// Mitsubishi GX Works2 project: BMA-PGM(V0.24)-20230412   PLC: Q06UDV

PROGRAM 02  // MANUAL
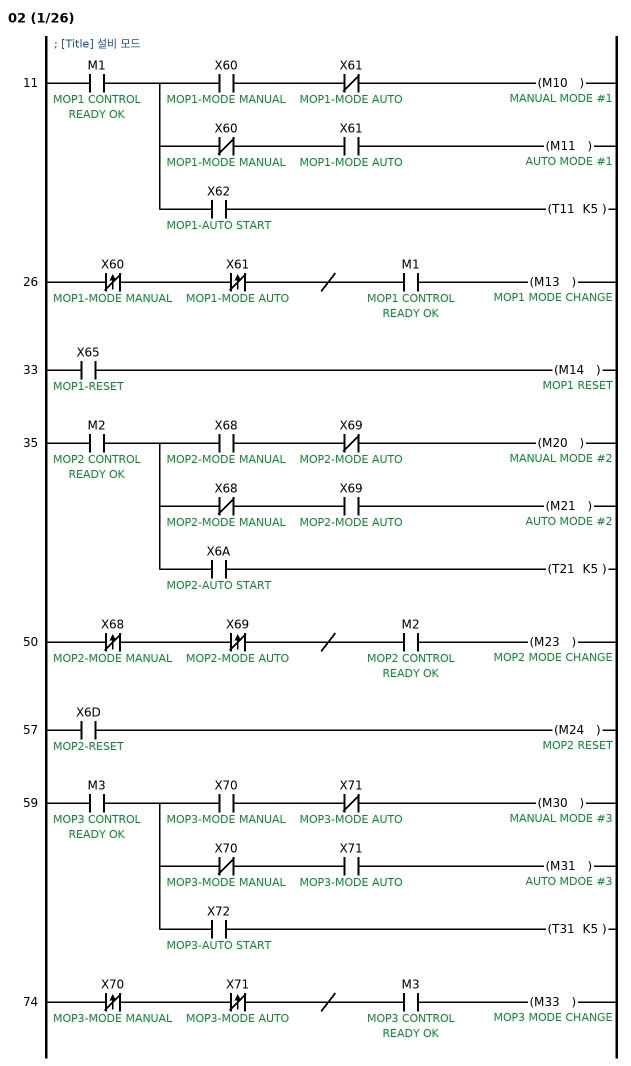
; [Title] 설비 모드
11    LD      M1  ; MOP1 CONTROL READY OK
      MPS
      AND     X60  ; MOP1-MODE MANUAL
      ANI     X61  ; MOP1-MODE AUTO
      OUT     M10  ; MANUAL MODE #1
      MRD
      ANI     X60  ; MOP1-MODE MANUAL
      AND     X61  ; MOP1-MODE AUTO
      OUT     M11  ; AUTO MODE #1
      MPP
      AND     X62  ; MOP1-AUTO START
      OUT     T11 K5
26    LDPI    X60  ; MOP1-MODE MANUAL
      ANDPI   X61  ; MOP1-MODE AUTO
      INV
      AND     M1  ; MOP1 CONTROL READY OK
      OUT     M13  ; MOP1 MODE CHANGE
33    LD      X65  ; MOP1-RESET
      OUT     M14  ; MOP1 RESET
35    LD      M2  ; MOP2 CONTROL READY OK
      MPS
      AND     X68  ; MOP2-MODE MANUAL
      ANI     X69  ; MOP2-MODE AUTO
      OUT     M20  ; MANUAL MODE #2
      MRD
      ANI     X68  ; MOP2-MODE MANUAL
      AND     X69  ; MOP2-MODE AUTO
      OUT     M21  ; AUTO MODE #2
      MPP
      AND     X6A  ; MOP2-AUTO START
      OUT     T21 K5
50    LDPI    X68  ; MOP2-MODE MANUAL
      ANDPI   X69  ; MOP2-MODE AUTO
      INV
      AND     M2  ; MOP2 CONTROL READY OK
      OUT     M23  ; MOP2 MODE CHANGE
57    LD      X6D  ; MOP2-RESET
      OUT     M24  ; MOP2 RESET
59    LD      M3  ; MOP3 CONTROL READY OK
      MPS
      AND     X70  ; MOP3-MODE MANUAL
      ANI     X71  ; MOP3-MODE AUTO
      OUT     M30  ; MANUAL MODE #3
      MRD
      ANI     X70  ; MOP3-MODE MANUAL
      AND     X71  ; MOP3-MODE AUTO
      OUT     M31  ; AUTO MDOE #3
      MPP
      AND     X72  ; MOP3-AUTO START
      OUT     T31 K5
74    LDPI    X70  ; MOP3-MODE MANUAL
      ANDPI   X71  ; MOP3-MODE AUTO
      INV
      AND     M3  ; MOP3 CONTROL READY OK
      OUT     M33  ; MOP3 MODE CHANGE
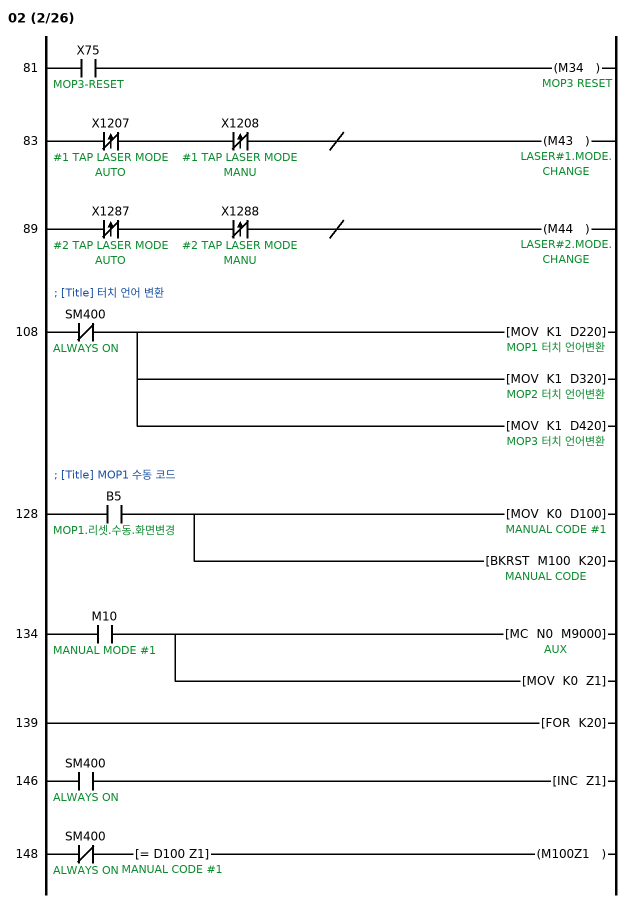
81    LD      X75  ; MOP3-RESET
      OUT     M34  ; MOP3 RESET
83    LDPI    X1207  ; #1 TAP LASER MODE AUTO
      ANDPI   X1208  ; #1 TAP LASER MODE MANU
      INV
      OUT     M43  ; LASER#1.MODE.CHANGE
89    LDPI    X1287  ; #2 TAP LASER MODE AUTO
      ANDPI   X1288  ; #2 TAP LASER MODE MANU
      INV
      OUT     M44  ; LASER#2.MODE.CHANGE
; [Title] 터치 언어 변환
108   LDI     SM400  ; ALWAYS ON
      MOV     K1 D220  ; MOP1 터치 언어변환
      MOV     K1 D320  ; MOP2 터치 언어변환
      MOV     K1 D420  ; MOP3 터치 언어변환
; [Title] MOP1 수동 코드
128   LD      B5  ; MOP1.리셋.수동.화면변경
      MOV     K0 D100  ; MANUAL CODE #1
      BKRST   M100 K20  ; MANUAL CODE
134   LD      M10  ; MANUAL MODE #1
      MC      N0 M9000  ; AUX
      MOV     K0 Z1
139   FOR     K20
        [note] 1~20
146   LD      SM400  ; ALWAYS ON
      INC     Z1
148   LDI     SM400  ; ALWAYS ON
      AND=    D100 Z1  ; MANUAL CODE #1
      OUT     M100Z1
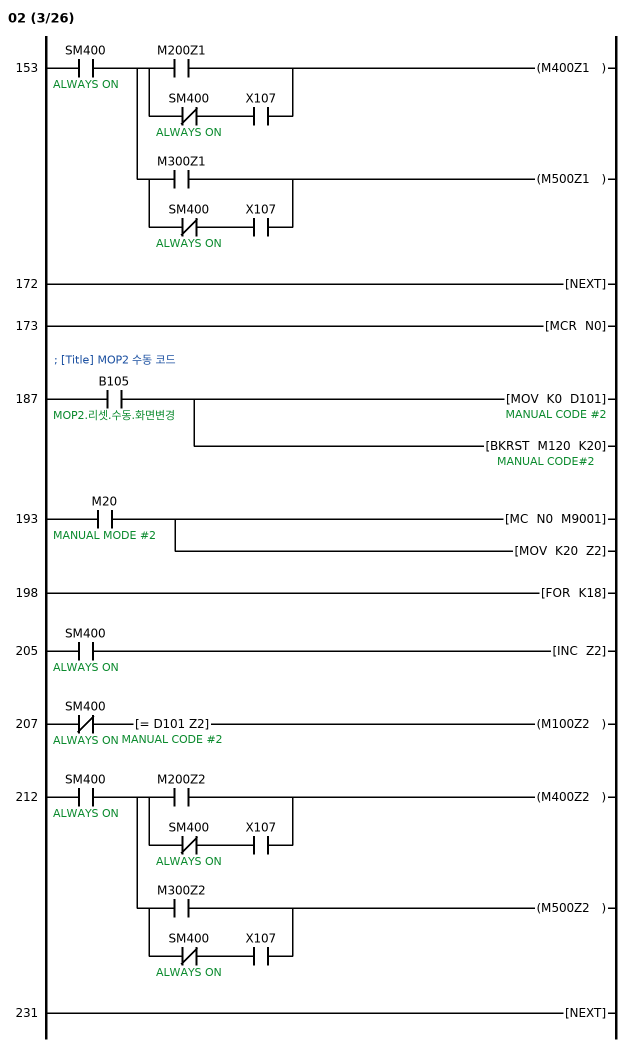
153   LD      SM400  ; ALWAYS ON
      MPS
      LD      M200Z1
      LDI     SM400  ; ALWAYS ON
      AND     X107
      ORB
      ANB
      OUT     M400Z1
      MPP
      LD      M300Z1
      LDI     SM400  ; ALWAYS ON
      AND     X107
      ORB
      ANB
      OUT     M500Z1
172   NEXT
173   MCR     N0
; [Title] MOP2 수동 코드
187   LD      B105  ; MOP2.리셋.수동.화면변경
      MOV     K0 D101  ; MANUAL CODE #2
      BKRST   M120 K20  ; MANUAL CODE#2
193   LD      M20  ; MANUAL MODE #2
      MC      N0 M9001
      MOV     K20 Z2
198   FOR     K18
        [note] 21~38
205   LD      SM400  ; ALWAYS ON
      INC     Z2
207   LDI     SM400  ; ALWAYS ON
      AND=    D101 Z2  ; MANUAL CODE #2
      OUT     M100Z2
212   LD      SM400  ; ALWAYS ON
      MPS
      LD      M200Z2
      LDI     SM400  ; ALWAYS ON
      AND     X107
      ORB
      ANB
      OUT     M400Z2
      MPP
      LD      M300Z2
      LDI     SM400  ; ALWAYS ON
      AND     X107
      ORB
      ANB
      OUT     M500Z2
231   NEXT
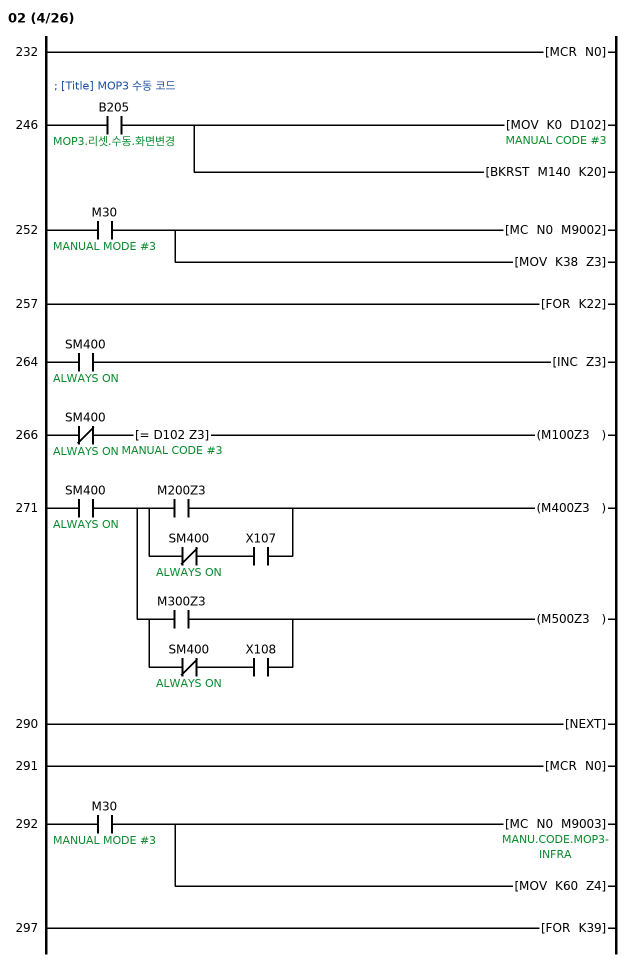
232   MCR     N0
; [Title] MOP3 수동 코드
246   LD      B205  ; MOP3.리셋.수동.화면변경
      MOV     K0 D102  ; MANUAL CODE #3
      BKRST   M140 K20
252   LD      M30  ; MANUAL MODE #3
      MC      N0 M9002
      MOV     K38 Z3
257   FOR     K22
        [note] 39~60
264   LD      SM400  ; ALWAYS ON
      INC     Z3
266   LDI     SM400  ; ALWAYS ON
      AND=    D102 Z3  ; MANUAL CODE #3
      OUT     M100Z3
271   LD      SM400  ; ALWAYS ON
      MPS
      LD      M200Z3
      LDI     SM400  ; ALWAYS ON
      AND     X107
      ORB
      ANB
      OUT     M400Z3
      MPP
      LD      M300Z3
      LDI     SM400  ; ALWAYS ON
      AND     X108
      ORB
      ANB
      OUT     M500Z3
290   NEXT
291   MCR     N0
292   LD      M30  ; MANUAL MODE #3
      MC      N0 M9003  ; MANU.CODE.MOP3-INFRA
      MOV     K60 Z4
297   FOR     K39
        [note] 61~99
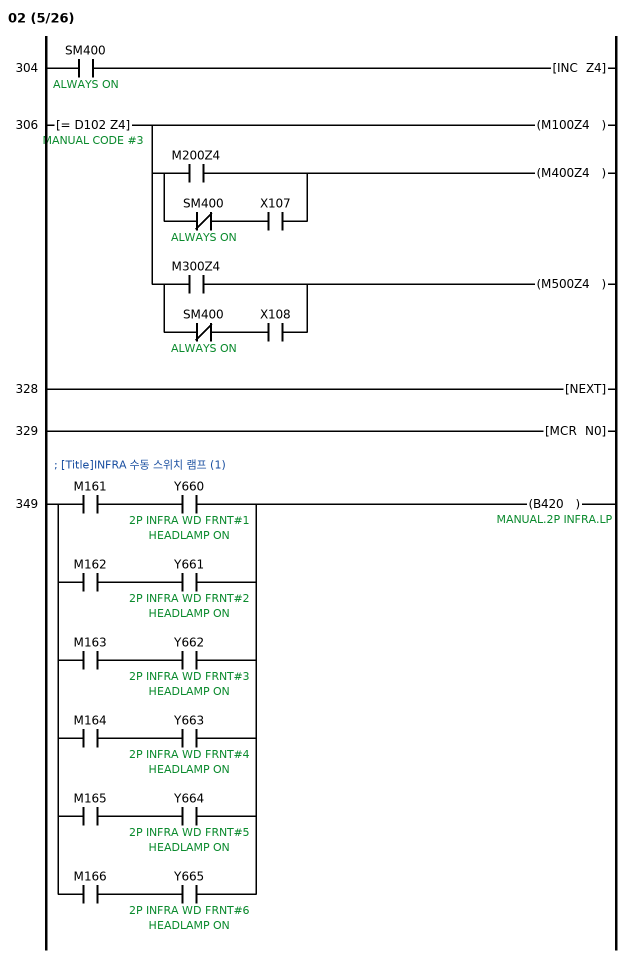
304   LD      SM400  ; ALWAYS ON
      INC     Z4
306   LD=     D102 Z4  ; MANUAL CODE #3
      OUT     M100Z4
      MPS
      LD      M200Z4
      LDI     SM400  ; ALWAYS ON
      AND     X107
      ORB
      ANB
      OUT     M400Z4
      MPP
      LD      M300Z4
      LDI     SM400  ; ALWAYS ON
      AND     X108
      ORB
      ANB
      OUT     M500Z4
328   NEXT
329   MCR     N0
; [Title]INFRA 수동 스위치 램프 (1)
349   LD      M161
      AND     Y660  ; 2P INFRA WD FRNT#1 HEADLAMP ON
      LD      M162
      AND     Y661  ; 2P INFRA WD FRNT#2 HEADLAMP ON
      ORB
      LD      M163
      AND     Y662  ; 2P INFRA WD FRNT#3 HEADLAMP ON
      ORB
      LD      M164
      AND     Y663  ; 2P INFRA WD FRNT#4 HEADLAMP ON
      ORB
      LD      M165
      AND     Y664  ; 2P INFRA WD FRNT#5 HEADLAMP ON
      ORB
      LD      M166
      AND     Y665  ; 2P INFRA WD FRNT#6 HEADLAMP ON
      ORB
      OUT     B420  ; MANUAL.2P INFRA.LP
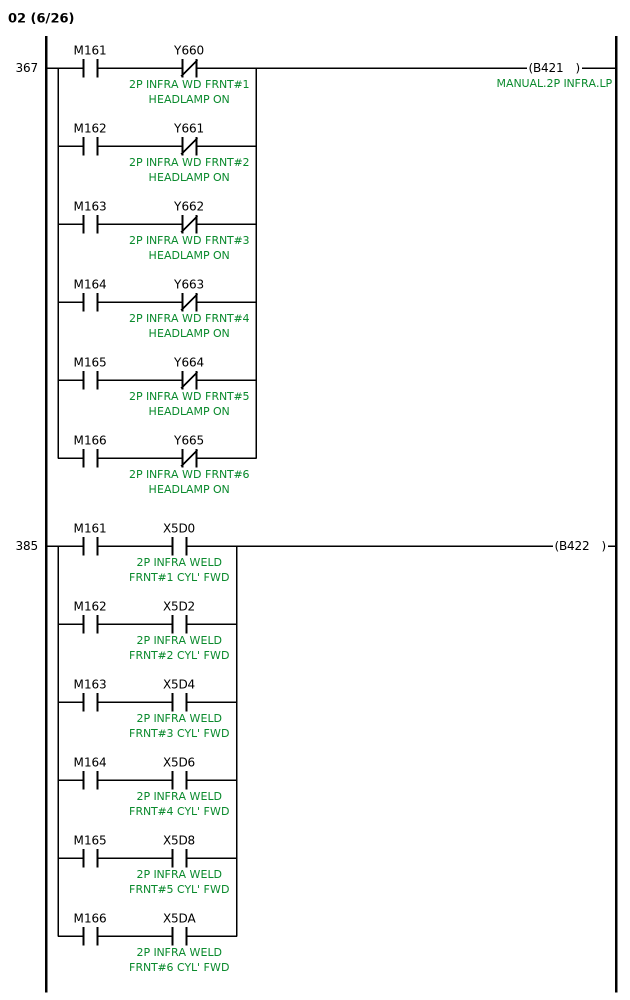
367   LD      M161
      ANI     Y660  ; 2P INFRA WD FRNT#1 HEADLAMP ON
      LD      M162
      ANI     Y661  ; 2P INFRA WD FRNT#2 HEADLAMP ON
      ORB
      LD      M163
      ANI     Y662  ; 2P INFRA WD FRNT#3 HEADLAMP ON
      ORB
      LD      M164
      ANI     Y663  ; 2P INFRA WD FRNT#4 HEADLAMP ON
      ORB
      LD      M165
      ANI     Y664  ; 2P INFRA WD FRNT#5 HEADLAMP ON
      ORB
      LD      M166
      ANI     Y665  ; 2P INFRA WD FRNT#6 HEADLAMP ON
      ORB
      OUT     B421  ; MANUAL.2P INFRA.LP
385   LD      M161
      AND     X5D0  ; 2P INFRA WELD FRNT#1 CYL' FWD
      LD      M162
      AND     X5D2  ; 2P INFRA WELD FRNT#2 CYL' FWD
      ORB
      LD      M163
      AND     X5D4  ; 2P INFRA WELD FRNT#3 CYL' FWD
      ORB
      LD      M164
      AND     X5D6  ; 2P INFRA WELD FRNT#4 CYL' FWD
      ORB
      LD      M165
      AND     X5D8  ; 2P INFRA WELD FRNT#5 CYL' FWD
      ORB
      LD      M166
      AND     X5DA  ; 2P INFRA WELD FRNT#6 CYL' FWD
      ORB
      OUT     B422
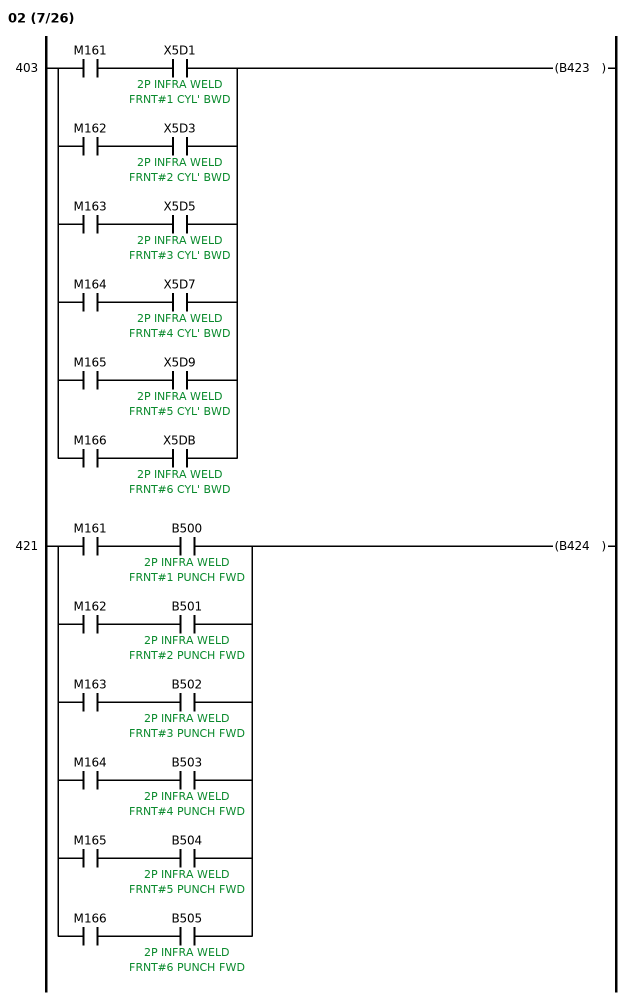
403   LD      M161
      AND     X5D1  ; 2P INFRA WELD FRNT#1 CYL' BWD
      LD      M162
      AND     X5D3  ; 2P INFRA WELD FRNT#2 CYL' BWD
      ORB
      LD      M163
      AND     X5D5  ; 2P INFRA WELD FRNT#3 CYL' BWD
      ORB
      LD      M164
      AND     X5D7  ; 2P INFRA WELD FRNT#4 CYL' BWD
      ORB
      LD      M165
      AND     X5D9  ; 2P INFRA WELD FRNT#5 CYL' BWD
      ORB
      LD      M166
      AND     X5DB  ; 2P INFRA WELD FRNT#6 CYL' BWD
      ORB
      OUT     B423
421   LD      M161
      AND     B500  ; 2P INFRA WELD FRNT#1 PUNCH FWD
      LD      M162
      AND     B501  ; 2P INFRA WELD FRNT#2 PUNCH FWD
      ORB
      LD      M163
      AND     B502  ; 2P INFRA WELD FRNT#3 PUNCH FWD
      ORB
      LD      M164
      AND     B503  ; 2P INFRA WELD FRNT#4 PUNCH FWD
      ORB
      LD      M165
      AND     B504  ; 2P INFRA WELD FRNT#5 PUNCH FWD
      ORB
      LD      M166
      AND     B505  ; 2P INFRA WELD FRNT#6 PUNCH FWD
      ORB
      OUT     B424
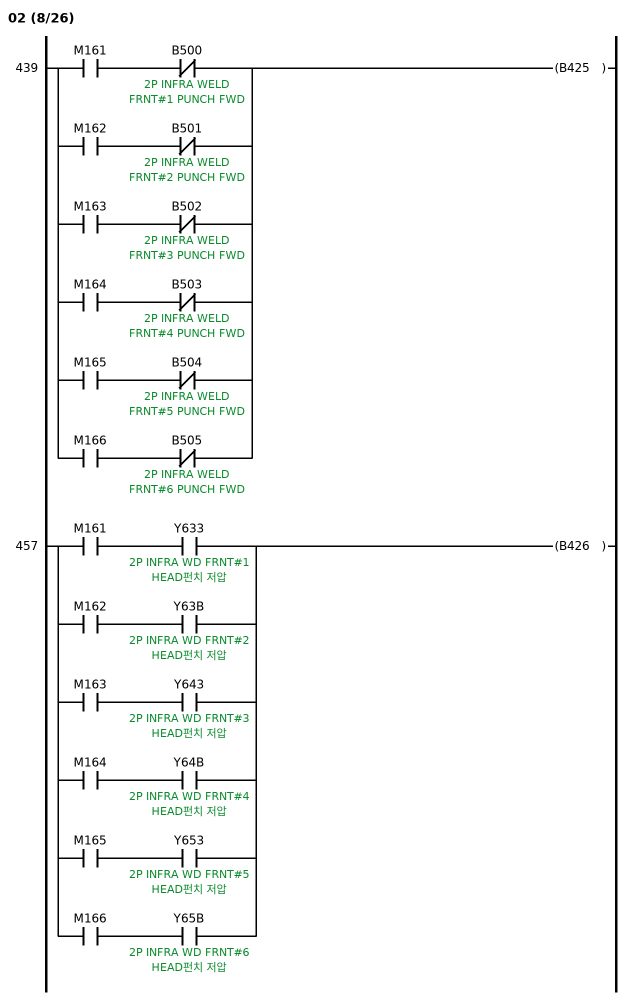
439   LD      M161
      ANI     B500  ; 2P INFRA WELD FRNT#1 PUNCH FWD
      LD      M162
      ANI     B501  ; 2P INFRA WELD FRNT#2 PUNCH FWD
      ORB
      LD      M163
      ANI     B502  ; 2P INFRA WELD FRNT#3 PUNCH FWD
      ORB
      LD      M164
      ANI     B503  ; 2P INFRA WELD FRNT#4 PUNCH FWD
      ORB
      LD      M165
      ANI     B504  ; 2P INFRA WELD FRNT#5 PUNCH FWD
      ORB
      LD      M166
      ANI     B505  ; 2P INFRA WELD FRNT#6 PUNCH FWD
      ORB
      OUT     B425
457   LD      M161
      AND     Y633  ; 2P INFRA WD FRNT#1 HEAD펀치 저압
      LD      M162
      AND     Y63B  ; 2P INFRA WD FRNT#2 HEAD펀치 저압
      ORB
      LD      M163
      AND     Y643  ; 2P INFRA WD FRNT#3 HEAD펀치 저압
      ORB
      LD      M164
      AND     Y64B  ; 2P INFRA WD FRNT#4 HEAD펀치 저압
      ORB
      LD      M165
      AND     Y653  ; 2P INFRA WD FRNT#5 HEAD펀치 저압
      ORB
      LD      M166
      AND     Y65B  ; 2P INFRA WD FRNT#6 HEAD펀치 저압
      ORB
      OUT     B426
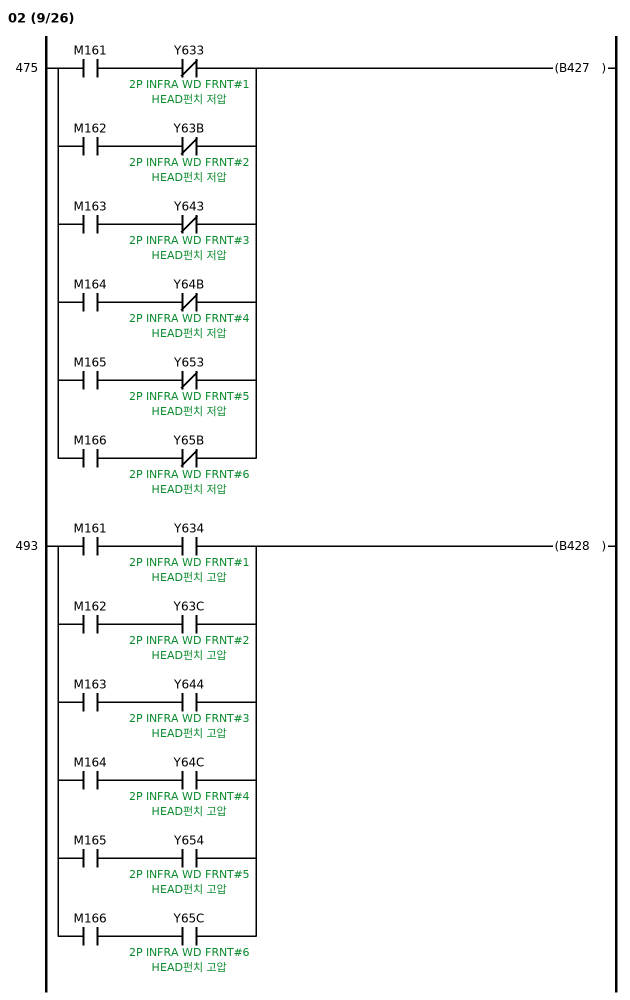
475   LD      M161
      ANI     Y633  ; 2P INFRA WD FRNT#1 HEAD펀치 저압
      LD      M162
      ANI     Y63B  ; 2P INFRA WD FRNT#2 HEAD펀치 저압
      ORB
      LD      M163
      ANI     Y643  ; 2P INFRA WD FRNT#3 HEAD펀치 저압
      ORB
      LD      M164
      ANI     Y64B  ; 2P INFRA WD FRNT#4 HEAD펀치 저압
      ORB
      LD      M165
      ANI     Y653  ; 2P INFRA WD FRNT#5 HEAD펀치 저압
      ORB
      LD      M166
      ANI     Y65B  ; 2P INFRA WD FRNT#6 HEAD펀치 저압
      ORB
      OUT     B427
493   LD      M161
      AND     Y634  ; 2P INFRA WD FRNT#1 HEAD펀치 고압
      LD      M162
      AND     Y63C  ; 2P INFRA WD FRNT#2 HEAD펀치 고압
      ORB
      LD      M163
      AND     Y644  ; 2P INFRA WD FRNT#3 HEAD펀치 고압
      ORB
      LD      M164
      AND     Y64C  ; 2P INFRA WD FRNT#4 HEAD펀치 고압
      ORB
      LD      M165
      AND     Y654  ; 2P INFRA WD FRNT#5 HEAD펀치 고압
      ORB
      LD      M166
      AND     Y65C  ; 2P INFRA WD FRNT#6 HEAD펀치 고압
      ORB
      OUT     B428
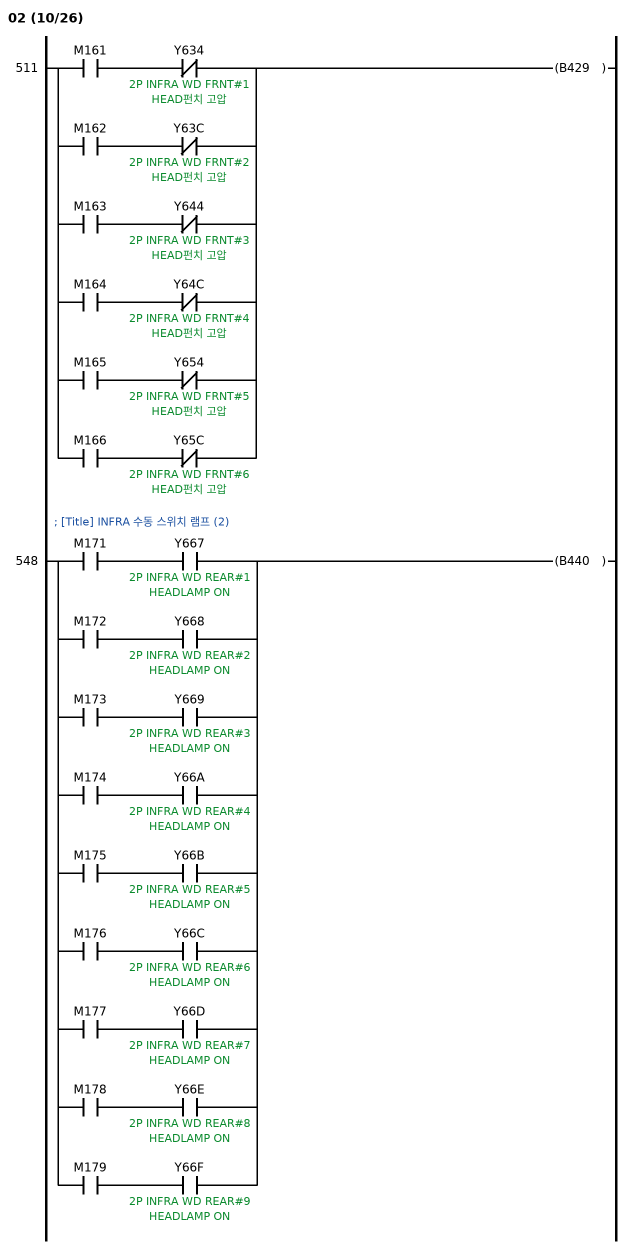
511   LD      M161
      ANI     Y634  ; 2P INFRA WD FRNT#1 HEAD펀치 고압
      LD      M162
      ANI     Y63C  ; 2P INFRA WD FRNT#2 HEAD펀치 고압
      ORB
      LD      M163
      ANI     Y644  ; 2P INFRA WD FRNT#3 HEAD펀치 고압
      ORB
      LD      M164
      ANI     Y64C  ; 2P INFRA WD FRNT#4 HEAD펀치 고압
      ORB
      LD      M165
      ANI     Y654  ; 2P INFRA WD FRNT#5 HEAD펀치 고압
      ORB
      LD      M166
      ANI     Y65C  ; 2P INFRA WD FRNT#6 HEAD펀치 고압
      ORB
      OUT     B429
; [Title] INFRA 수동 스위치 램프 (2)
548   LD      M171
      AND     Y667  ; 2P INFRA WD REAR#1 HEADLAMP ON
      LD      M172
      AND     Y668  ; 2P INFRA WD REAR#2 HEADLAMP ON
      ORB
      LD      M173
      AND     Y669  ; 2P INFRA WD REAR#3 HEADLAMP ON
      ORB
      LD      M174
      AND     Y66A  ; 2P INFRA WD REAR#4 HEADLAMP ON
      ORB
      LD      M175
      AND     Y66B  ; 2P INFRA WD REAR#5 HEADLAMP ON
      ORB
      LD      M176
      AND     Y66C  ; 2P INFRA WD REAR#6 HEADLAMP ON
      ORB
      LD      M177
      AND     Y66D  ; 2P INFRA WD REAR#7 HEADLAMP ON
      ORB
      LD      M178
      AND     Y66E  ; 2P INFRA WD REAR#8 HEADLAMP ON
      ORB
      LD      M179
      AND     Y66F  ; 2P INFRA WD REAR#9 HEADLAMP ON
      ORB
      OUT     B440
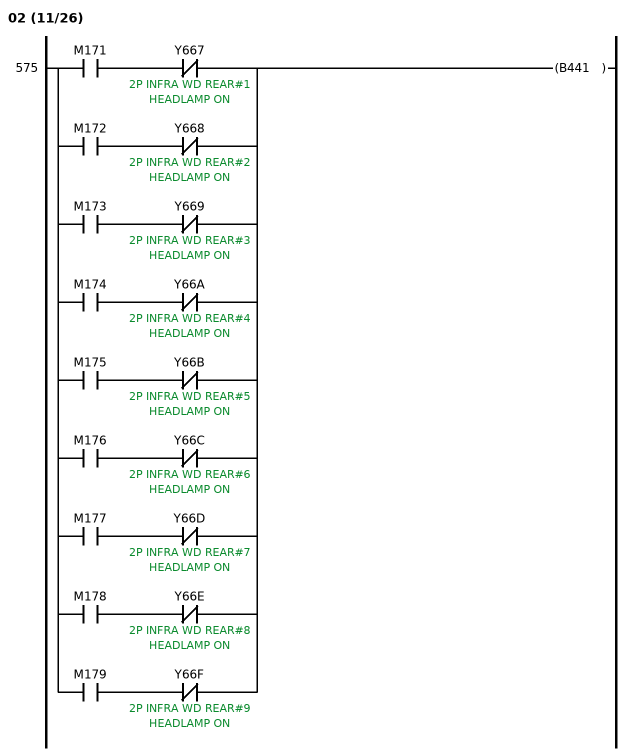
575   LD      M171
      ANI     Y667  ; 2P INFRA WD REAR#1 HEADLAMP ON
      LD      M172
      ANI     Y668  ; 2P INFRA WD REAR#2 HEADLAMP ON
      ORB
      LD      M173
      ANI     Y669  ; 2P INFRA WD REAR#3 HEADLAMP ON
      ORB
      LD      M174
      ANI     Y66A  ; 2P INFRA WD REAR#4 HEADLAMP ON
      ORB
      LD      M175
      ANI     Y66B  ; 2P INFRA WD REAR#5 HEADLAMP ON
      ORB
      LD      M176
      ANI     Y66C  ; 2P INFRA WD REAR#6 HEADLAMP ON
      ORB
      LD      M177
      ANI     Y66D  ; 2P INFRA WD REAR#7 HEADLAMP ON
      ORB
      LD      M178
      ANI     Y66E  ; 2P INFRA WD REAR#8 HEADLAMP ON
      ORB
      LD      M179
      ANI     Y66F  ; 2P INFRA WD REAR#9 HEADLAMP ON
      ORB
      OUT     B441
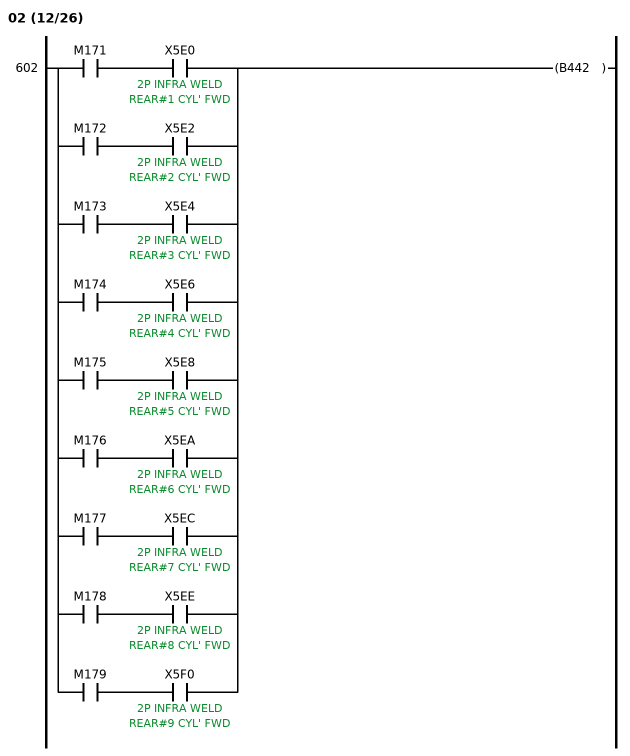
602   LD      M171
      AND     X5E0  ; 2P INFRA WELD REAR#1 CYL' FWD
      LD      M172
      AND     X5E2  ; 2P INFRA WELD REAR#2 CYL' FWD
      ORB
      LD      M173
      AND     X5E4  ; 2P INFRA WELD REAR#3 CYL' FWD
      ORB
      LD      M174
      AND     X5E6  ; 2P INFRA WELD REAR#4 CYL' FWD
      ORB
      LD      M175
      AND     X5E8  ; 2P INFRA WELD REAR#5 CYL' FWD
      ORB
      LD      M176
      AND     X5EA  ; 2P INFRA WELD REAR#6 CYL' FWD
      ORB
      LD      M177
      AND     X5EC  ; 2P INFRA WELD REAR#7 CYL' FWD
      ORB
      LD      M178
      AND     X5EE  ; 2P INFRA WELD REAR#8 CYL' FWD
      ORB
      LD      M179
      AND     X5F0  ; 2P INFRA WELD REAR#9 CYL' FWD
      ORB
      OUT     B442
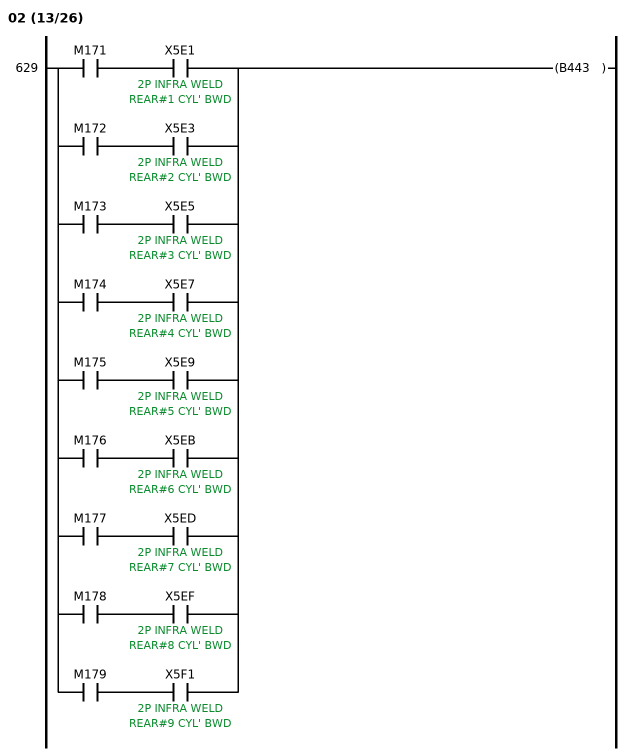
629   LD      M171
      AND     X5E1  ; 2P INFRA WELD REAR#1 CYL' BWD
      LD      M172
      AND     X5E3  ; 2P INFRA WELD REAR#2 CYL' BWD
      ORB
      LD      M173
      AND     X5E5  ; 2P INFRA WELD REAR#3 CYL' BWD
      ORB
      LD      M174
      AND     X5E7  ; 2P INFRA WELD REAR#4 CYL' BWD
      ORB
      LD      M175
      AND     X5E9  ; 2P INFRA WELD REAR#5 CYL' BWD
      ORB
      LD      M176
      AND     X5EB  ; 2P INFRA WELD REAR#6 CYL' BWD
      ORB
      LD      M177
      AND     X5ED  ; 2P INFRA WELD REAR#7 CYL' BWD
      ORB
      LD      M178
      AND     X5EF  ; 2P INFRA WELD REAR#8 CYL' BWD
      ORB
      LD      M179
      AND     X5F1  ; 2P INFRA WELD REAR#9 CYL' BWD
      ORB
      OUT     B443
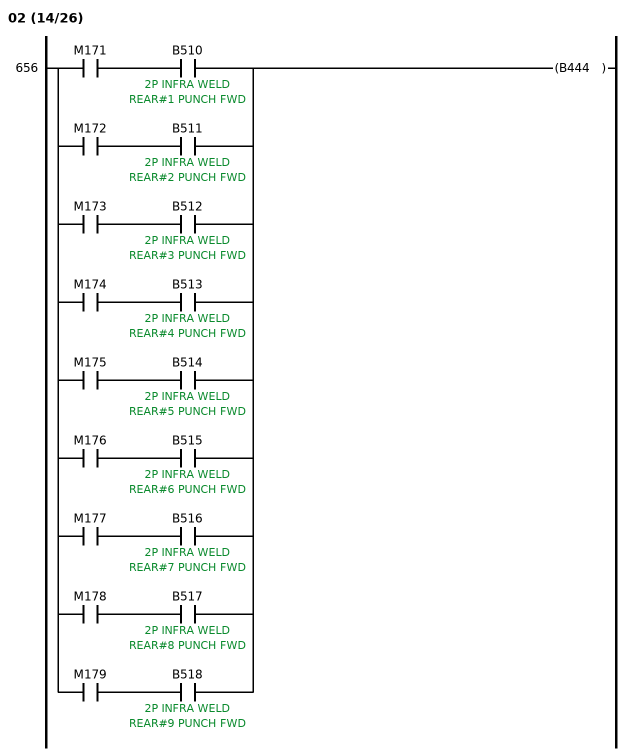
656   LD      M171
      AND     B510  ; 2P INFRA WELD REAR#1 PUNCH FWD
      LD      M172
      AND     B511  ; 2P INFRA WELD REAR#2 PUNCH FWD
      ORB
      LD      M173
      AND     B512  ; 2P INFRA WELD REAR#3 PUNCH FWD
      ORB
      LD      M174
      AND     B513  ; 2P INFRA WELD REAR#4 PUNCH FWD
      ORB
      LD      M175
      AND     B514  ; 2P INFRA WELD REAR#5 PUNCH FWD
      ORB
      LD      M176
      AND     B515  ; 2P INFRA WELD REAR#6 PUNCH FWD
      ORB
      LD      M177
      AND     B516  ; 2P INFRA WELD REAR#7 PUNCH FWD
      ORB
      LD      M178
      AND     B517  ; 2P INFRA WELD REAR#8 PUNCH FWD
      ORB
      LD      M179
      AND     B518  ; 2P INFRA WELD REAR#9 PUNCH FWD
      ORB
      OUT     B444
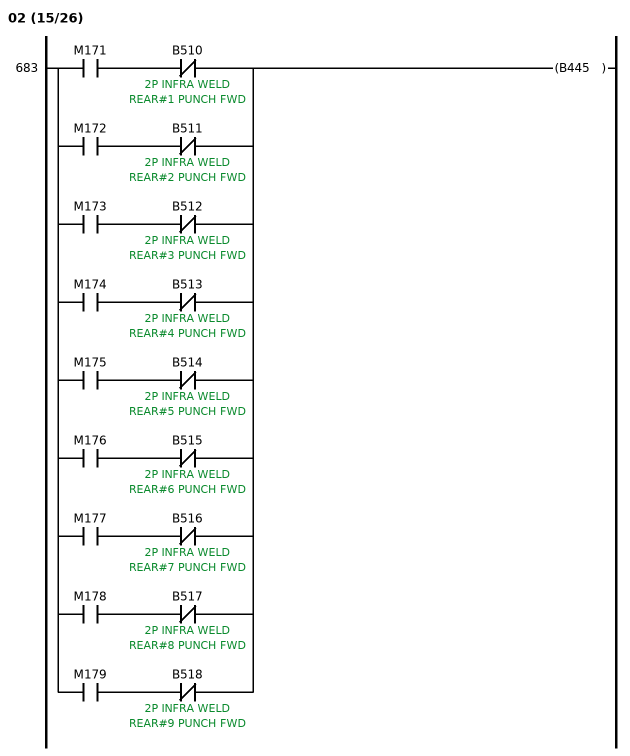
683   LD      M171
      ANI     B510  ; 2P INFRA WELD REAR#1 PUNCH FWD
      LD      M172
      ANI     B511  ; 2P INFRA WELD REAR#2 PUNCH FWD
      ORB
      LD      M173
      ANI     B512  ; 2P INFRA WELD REAR#3 PUNCH FWD
      ORB
      LD      M174
      ANI     B513  ; 2P INFRA WELD REAR#4 PUNCH FWD
      ORB
      LD      M175
      ANI     B514  ; 2P INFRA WELD REAR#5 PUNCH FWD
      ORB
      LD      M176
      ANI     B515  ; 2P INFRA WELD REAR#6 PUNCH FWD
      ORB
      LD      M177
      ANI     B516  ; 2P INFRA WELD REAR#7 PUNCH FWD
      ORB
      LD      M178
      ANI     B517  ; 2P INFRA WELD REAR#8 PUNCH FWD
      ORB
      LD      M179
      ANI     B518  ; 2P INFRA WELD REAR#9 PUNCH FWD
      ORB
      OUT     B445
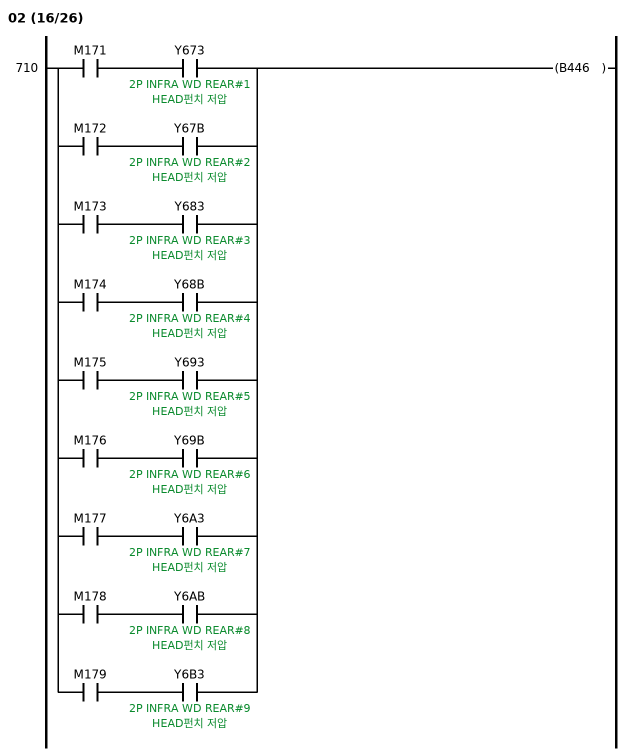
710   LD      M171
      AND     Y673  ; 2P INFRA WD REAR#1 HEAD펀치 저압
      LD      M172
      AND     Y67B  ; 2P INFRA WD REAR#2 HEAD펀치 저압
      ORB
      LD      M173
      AND     Y683  ; 2P INFRA WD REAR#3 HEAD펀치 저압
      ORB
      LD      M174
      AND     Y68B  ; 2P INFRA WD REAR#4 HEAD펀치 저압
      ORB
      LD      M175
      AND     Y693  ; 2P INFRA WD REAR#5 HEAD펀치 저압
      ORB
      LD      M176
      AND     Y69B  ; 2P INFRA WD REAR#6 HEAD펀치 저압
      ORB
      LD      M177
      AND     Y6A3  ; 2P INFRA WD REAR#7 HEAD펀치 저압
      ORB
      LD      M178
      AND     Y6AB  ; 2P INFRA WD REAR#8 HEAD펀치 저압
      ORB
      LD      M179
      AND     Y6B3  ; 2P INFRA WD REAR#9 HEAD펀치 저압
      ORB
      OUT     B446
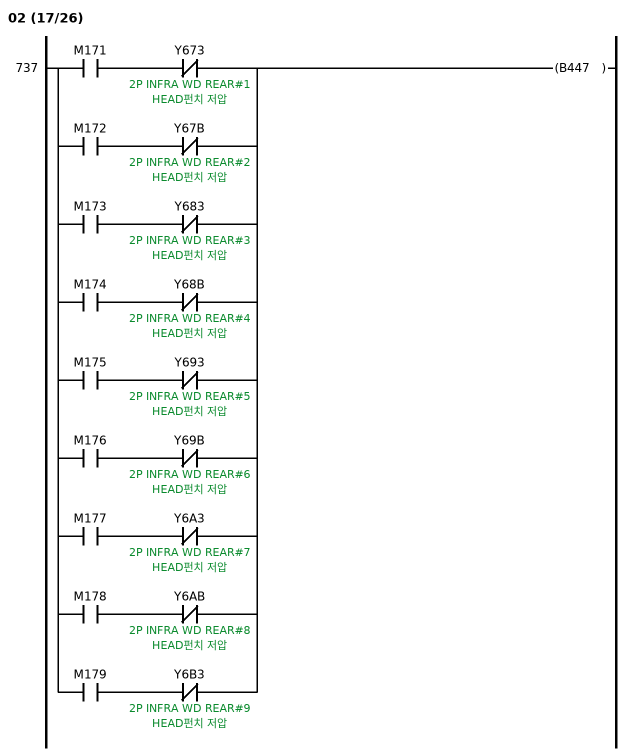
737   LD      M171
      ANI     Y673  ; 2P INFRA WD REAR#1 HEAD펀치 저압
      LD      M172
      ANI     Y67B  ; 2P INFRA WD REAR#2 HEAD펀치 저압
      ORB
      LD      M173
      ANI     Y683  ; 2P INFRA WD REAR#3 HEAD펀치 저압
      ORB
      LD      M174
      ANI     Y68B  ; 2P INFRA WD REAR#4 HEAD펀치 저압
      ORB
      LD      M175
      ANI     Y693  ; 2P INFRA WD REAR#5 HEAD펀치 저압
      ORB
      LD      M176
      ANI     Y69B  ; 2P INFRA WD REAR#6 HEAD펀치 저압
      ORB
      LD      M177
      ANI     Y6A3  ; 2P INFRA WD REAR#7 HEAD펀치 저압
      ORB
      LD      M178
      ANI     Y6AB  ; 2P INFRA WD REAR#8 HEAD펀치 저압
      ORB
      LD      M179
      ANI     Y6B3  ; 2P INFRA WD REAR#9 HEAD펀치 저압
      ORB
      OUT     B447
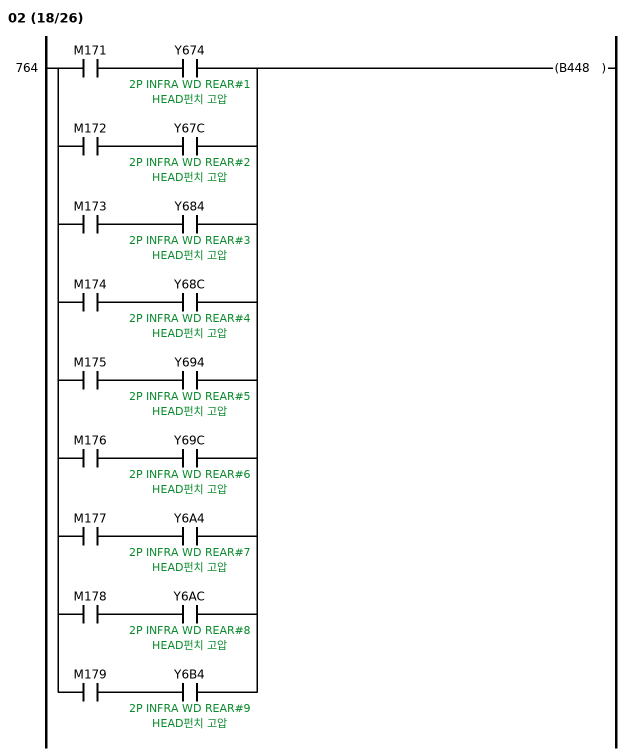
764   LD      M171
      AND     Y674  ; 2P INFRA WD REAR#1 HEAD펀치 고압
      LD      M172
      AND     Y67C  ; 2P INFRA WD REAR#2 HEAD펀치 고압
      ORB
      LD      M173
      AND     Y684  ; 2P INFRA WD REAR#3 HEAD펀치 고압
      ORB
      LD      M174
      AND     Y68C  ; 2P INFRA WD REAR#4 HEAD펀치 고압
      ORB
      LD      M175
      AND     Y694  ; 2P INFRA WD REAR#5 HEAD펀치 고압
      ORB
      LD      M176
      AND     Y69C  ; 2P INFRA WD REAR#6 HEAD펀치 고압
      ORB
      LD      M177
      AND     Y6A4  ; 2P INFRA WD REAR#7 HEAD펀치 고압
      ORB
      LD      M178
      AND     Y6AC  ; 2P INFRA WD REAR#8 HEAD펀치 고압
      ORB
      LD      M179
      AND     Y6B4  ; 2P INFRA WD REAR#9 HEAD펀치 고압
      ORB
      OUT     B448
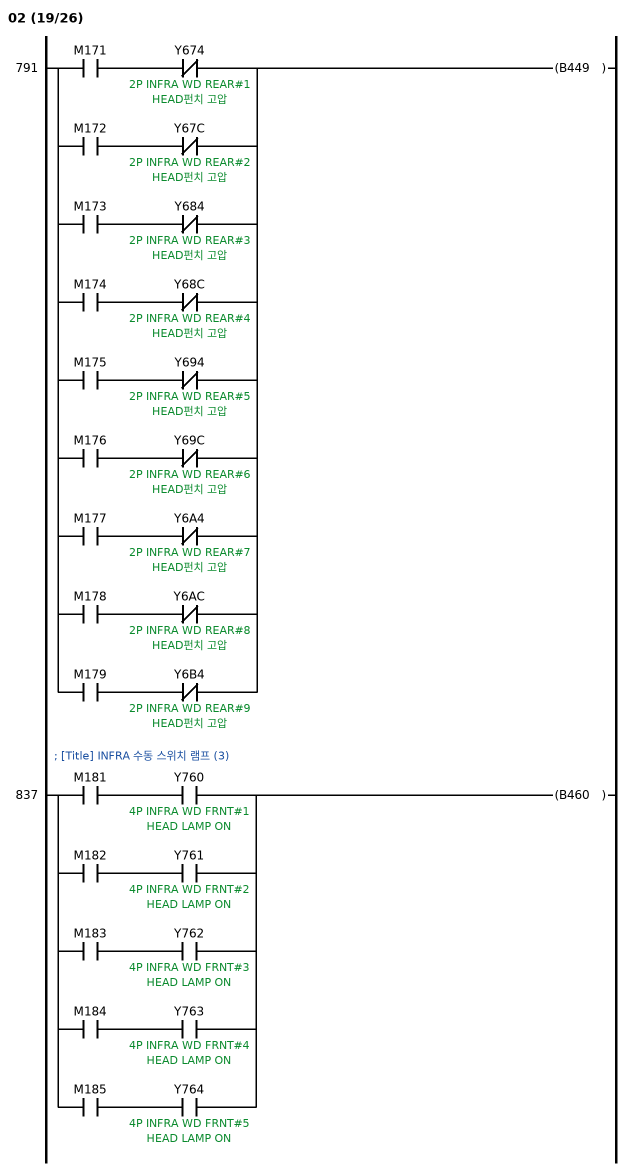
791   LD      M171
      ANI     Y674  ; 2P INFRA WD REAR#1 HEAD펀치 고압
      LD      M172
      ANI     Y67C  ; 2P INFRA WD REAR#2 HEAD펀치 고압
      ORB
      LD      M173
      ANI     Y684  ; 2P INFRA WD REAR#3 HEAD펀치 고압
      ORB
      LD      M174
      ANI     Y68C  ; 2P INFRA WD REAR#4 HEAD펀치 고압
      ORB
      LD      M175
      ANI     Y694  ; 2P INFRA WD REAR#5 HEAD펀치 고압
      ORB
      LD      M176
      ANI     Y69C  ; 2P INFRA WD REAR#6 HEAD펀치 고압
      ORB
      LD      M177
      ANI     Y6A4  ; 2P INFRA WD REAR#7 HEAD펀치 고압
      ORB
      LD      M178
      ANI     Y6AC  ; 2P INFRA WD REAR#8 HEAD펀치 고압
      ORB
      LD      M179
      ANI     Y6B4  ; 2P INFRA WD REAR#9 HEAD펀치 고압
      ORB
      OUT     B449
; [Title] INFRA 수동 스위치 램프 (3)
837   LD      M181
      AND     Y760  ; 4P INFRA WD FRNT#1 HEAD LAMP ON
      LD      M182
      AND     Y761  ; 4P INFRA WD FRNT#2 HEAD LAMP ON
      ORB
      LD      M183
      AND     Y762  ; 4P INFRA WD FRNT#3 HEAD LAMP ON
      ORB
      LD      M184
      AND     Y763  ; 4P INFRA WD FRNT#4 HEAD LAMP ON
      ORB
      LD      M185
      AND     Y764  ; 4P INFRA WD FRNT#5 HEAD LAMP ON
      ORB
      OUT     B460
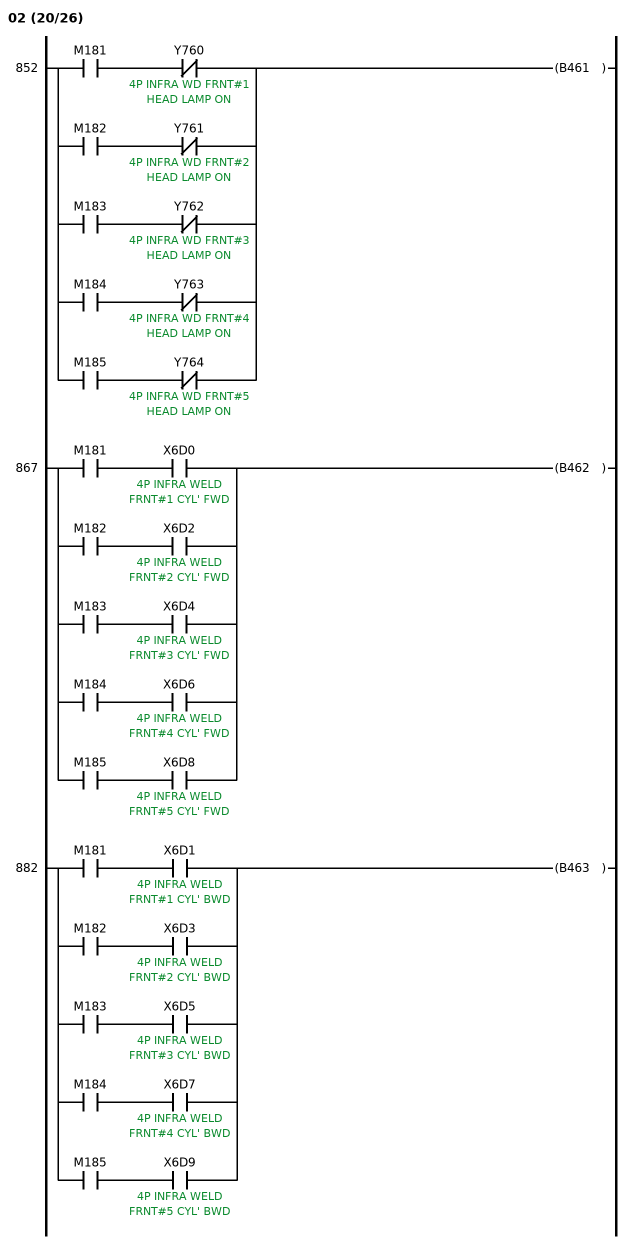
852   LD      M181
      ANI     Y760  ; 4P INFRA WD FRNT#1 HEAD LAMP ON
      LD      M182
      ANI     Y761  ; 4P INFRA WD FRNT#2 HEAD LAMP ON
      ORB
      LD      M183
      ANI     Y762  ; 4P INFRA WD FRNT#3 HEAD LAMP ON
      ORB
      LD      M184
      ANI     Y763  ; 4P INFRA WD FRNT#4 HEAD LAMP ON
      ORB
      LD      M185
      ANI     Y764  ; 4P INFRA WD FRNT#5 HEAD LAMP ON
      ORB
      OUT     B461
867   LD      M181
      AND     X6D0  ; 4P INFRA WELD FRNT#1 CYL' FWD
      LD      M182
      AND     X6D2  ; 4P INFRA WELD FRNT#2 CYL' FWD
      ORB
      LD      M183
      AND     X6D4  ; 4P INFRA WELD FRNT#3 CYL' FWD
      ORB
      LD      M184
      AND     X6D6  ; 4P INFRA WELD FRNT#4 CYL' FWD
      ORB
      LD      M185
      AND     X6D8  ; 4P INFRA WELD FRNT#5 CYL' FWD
      ORB
      OUT     B462
882   LD      M181
      AND     X6D1  ; 4P INFRA WELD FRNT#1 CYL' BWD
      LD      M182
      AND     X6D3  ; 4P INFRA WELD FRNT#2 CYL' BWD
      ORB
      LD      M183
      AND     X6D5  ; 4P INFRA WELD FRNT#3 CYL' BWD
      ORB
      LD      M184
      AND     X6D7  ; 4P INFRA WELD FRNT#4 CYL' BWD
      ORB
      LD      M185
      AND     X6D9  ; 4P INFRA WELD FRNT#5 CYL' BWD
      ORB
      OUT     B463
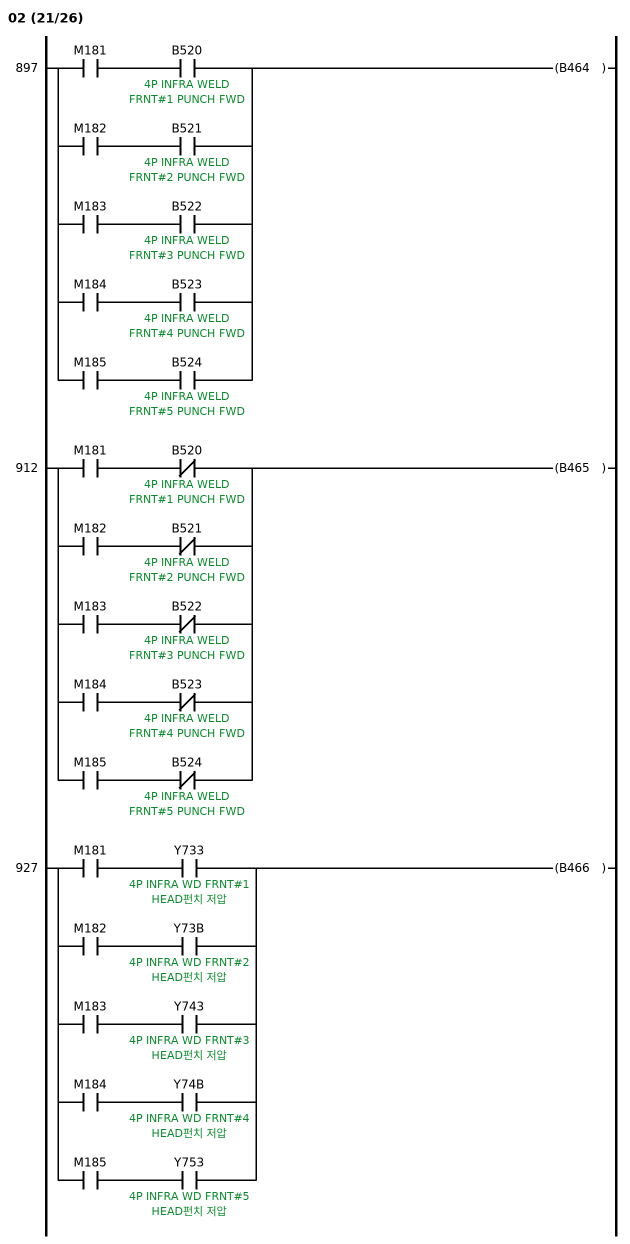
897   LD      M181
      AND     B520  ; 4P INFRA WELD FRNT#1 PUNCH FWD
      LD      M182
      AND     B521  ; 4P INFRA WELD FRNT#2 PUNCH FWD
      ORB
      LD      M183
      AND     B522  ; 4P INFRA WELD FRNT#3 PUNCH FWD
      ORB
      LD      M184
      AND     B523  ; 4P INFRA WELD FRNT#4 PUNCH FWD
      ORB
      LD      M185
      AND     B524  ; 4P INFRA WELD FRNT#5 PUNCH FWD
      ORB
      OUT     B464
912   LD      M181
      ANI     B520  ; 4P INFRA WELD FRNT#1 PUNCH FWD
      LD      M182
      ANI     B521  ; 4P INFRA WELD FRNT#2 PUNCH FWD
      ORB
      LD      M183
      ANI     B522  ; 4P INFRA WELD FRNT#3 PUNCH FWD
      ORB
      LD      M184
      ANI     B523  ; 4P INFRA WELD FRNT#4 PUNCH FWD
      ORB
      LD      M185
      ANI     B524  ; 4P INFRA WELD FRNT#5 PUNCH FWD
      ORB
      OUT     B465
927   LD      M181
      AND     Y733  ; 4P INFRA WD FRNT#1 HEAD펀치 저압
      LD      M182
      AND     Y73B  ; 4P INFRA WD FRNT#2 HEAD펀치 저압
      ORB
      LD      M183
      AND     Y743  ; 4P INFRA WD FRNT#3 HEAD펀치 저압
      ORB
      LD      M184
      AND     Y74B  ; 4P INFRA WD FRNT#4 HEAD펀치 저압
      ORB
      LD      M185
      AND     Y753  ; 4P INFRA WD FRNT#5 HEAD펀치 저압
      ORB
      OUT     B466
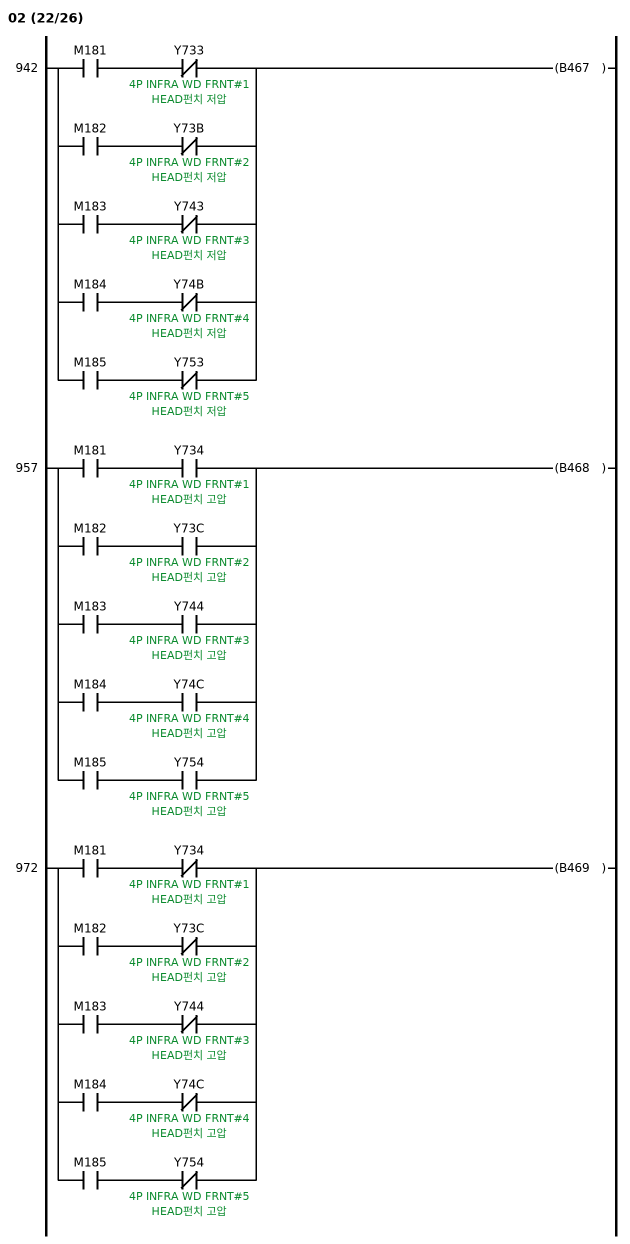
942   LD      M181
      ANI     Y733  ; 4P INFRA WD FRNT#1 HEAD펀치 저압
      LD      M182
      ANI     Y73B  ; 4P INFRA WD FRNT#2 HEAD펀치 저압
      ORB
      LD      M183
      ANI     Y743  ; 4P INFRA WD FRNT#3 HEAD펀치 저압
      ORB
      LD      M184
      ANI     Y74B  ; 4P INFRA WD FRNT#4 HEAD펀치 저압
      ORB
      LD      M185
      ANI     Y753  ; 4P INFRA WD FRNT#5 HEAD펀치 저압
      ORB
      OUT     B467
957   LD      M181
      AND     Y734  ; 4P INFRA WD FRNT#1 HEAD펀치 고압
      LD      M182
      AND     Y73C  ; 4P INFRA WD FRNT#2 HEAD펀치 고압
      ORB
      LD      M183
      AND     Y744  ; 4P INFRA WD FRNT#3 HEAD펀치 고압
      ORB
      LD      M184
      AND     Y74C  ; 4P INFRA WD FRNT#4 HEAD펀치 고압
      ORB
      LD      M185
      AND     Y754  ; 4P INFRA WD FRNT#5 HEAD펀치 고압
      ORB
      OUT     B468
972   LD      M181
      ANI     Y734  ; 4P INFRA WD FRNT#1 HEAD펀치 고압
      LD      M182
      ANI     Y73C  ; 4P INFRA WD FRNT#2 HEAD펀치 고압
      ORB
      LD      M183
      ANI     Y744  ; 4P INFRA WD FRNT#3 HEAD펀치 고압
      ORB
      LD      M184
      ANI     Y74C  ; 4P INFRA WD FRNT#4 HEAD펀치 고압
      ORB
      LD      M185
      ANI     Y754  ; 4P INFRA WD FRNT#5 HEAD펀치 고압
      ORB
      OUT     B469
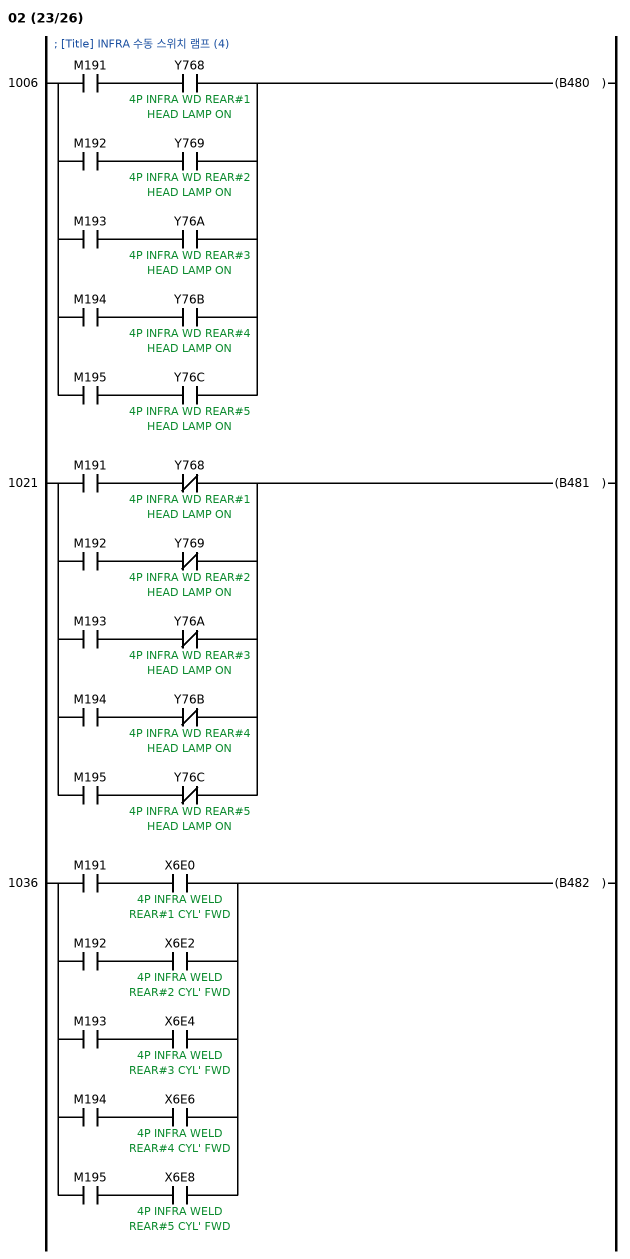
; [Title] INFRA 수동 스위치 램프 (4)
1006  LD      M191
      AND     Y768  ; 4P INFRA WD REAR#1 HEAD LAMP ON
      LD      M192
      AND     Y769  ; 4P INFRA WD REAR#2 HEAD LAMP ON
      ORB
      LD      M193
      AND     Y76A  ; 4P INFRA WD REAR#3 HEAD LAMP ON
      ORB
      LD      M194
      AND     Y76B  ; 4P INFRA WD REAR#4 HEAD LAMP ON
      ORB
      LD      M195
      AND     Y76C  ; 4P INFRA WD REAR#5 HEAD LAMP ON
      ORB
      OUT     B480
1021  LD      M191
      ANI     Y768  ; 4P INFRA WD REAR#1 HEAD LAMP ON
      LD      M192
      ANI     Y769  ; 4P INFRA WD REAR#2 HEAD LAMP ON
      ORB
      LD      M193
      ANI     Y76A  ; 4P INFRA WD REAR#3 HEAD LAMP ON
      ORB
      LD      M194
      ANI     Y76B  ; 4P INFRA WD REAR#4 HEAD LAMP ON
      ORB
      LD      M195
      ANI     Y76C  ; 4P INFRA WD REAR#5 HEAD LAMP ON
      ORB
      OUT     B481
1036  LD      M191
      AND     X6E0  ; 4P INFRA WELD REAR#1 CYL' FWD
      LD      M192
      AND     X6E2  ; 4P INFRA WELD REAR#2 CYL' FWD
      ORB
      LD      M193
      AND     X6E4  ; 4P INFRA WELD REAR#3 CYL' FWD
      ORB
      LD      M194
      AND     X6E6  ; 4P INFRA WELD REAR#4 CYL' FWD
      ORB
      LD      M195
      AND     X6E8  ; 4P INFRA WELD REAR#5 CYL' FWD
      ORB
      OUT     B482
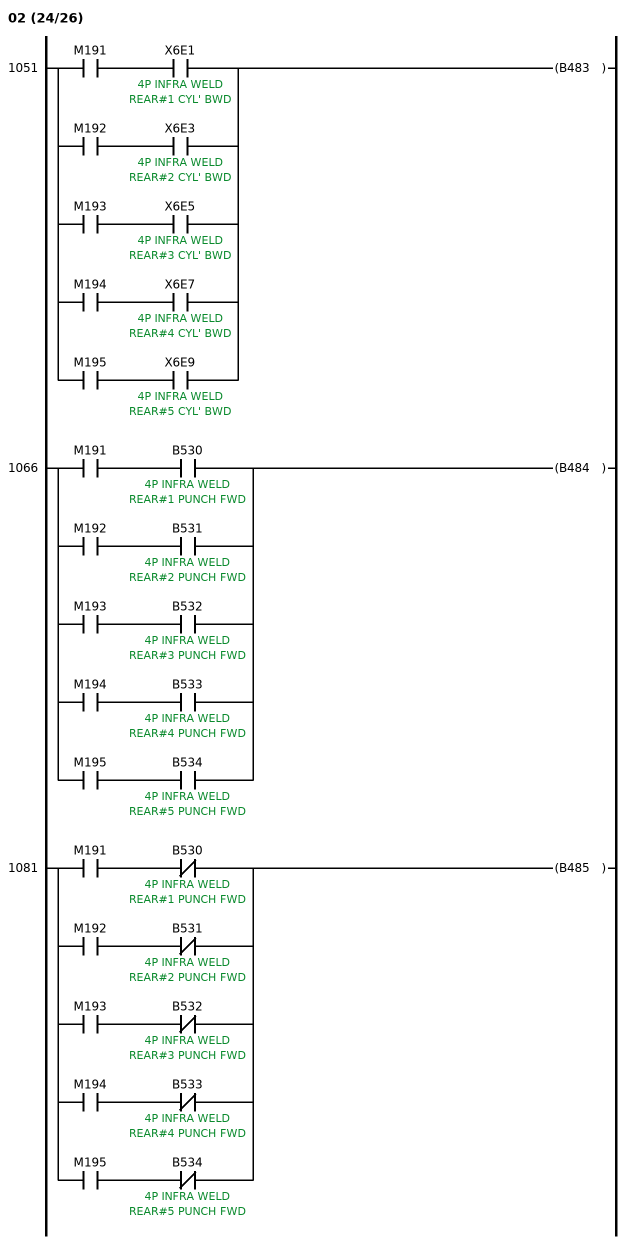
1051  LD      M191
      AND     X6E1  ; 4P INFRA WELD REAR#1 CYL' BWD
      LD      M192
      AND     X6E3  ; 4P INFRA WELD REAR#2 CYL' BWD
      ORB
      LD      M193
      AND     X6E5  ; 4P INFRA WELD REAR#3 CYL' BWD
      ORB
      LD      M194
      AND     X6E7  ; 4P INFRA WELD REAR#4 CYL' BWD
      ORB
      LD      M195
      AND     X6E9  ; 4P INFRA WELD REAR#5 CYL' BWD
      ORB
      OUT     B483
1066  LD      M191
      AND     B530  ; 4P INFRA WELD REAR#1 PUNCH FWD
      LD      M192
      AND     B531  ; 4P INFRA WELD REAR#2 PUNCH FWD
      ORB
      LD      M193
      AND     B532  ; 4P INFRA WELD REAR#3 PUNCH FWD
      ORB
      LD      M194
      AND     B533  ; 4P INFRA WELD REAR#4 PUNCH FWD
      ORB
      LD      M195
      AND     B534  ; 4P INFRA WELD REAR#5 PUNCH FWD
      ORB
      OUT     B484
1081  LD      M191
      ANI     B530  ; 4P INFRA WELD REAR#1 PUNCH FWD
      LD      M192
      ANI     B531  ; 4P INFRA WELD REAR#2 PUNCH FWD
      ORB
      LD      M193
      ANI     B532  ; 4P INFRA WELD REAR#3 PUNCH FWD
      ORB
      LD      M194
      ANI     B533  ; 4P INFRA WELD REAR#4 PUNCH FWD
      ORB
      LD      M195
      ANI     B534  ; 4P INFRA WELD REAR#5 PUNCH FWD
      ORB
      OUT     B485
